% RSLogix 500 project COMPARATOR_BAK026.RSS, saved by version 8.30.00.16 %
PROJECT "UNTITLED"    % processor: Bul.1763 MicroLogix 1100 Series B %

PROGRAM FILES
  LAD 2   9 rungs

DATA FILES
  O0 OUTPUT  4 elements
  I1 INPUT  6 elements
  S2 STATUS  66 elements
  B3 BINARY  1 elements
  T4 TIMER  1 elements
  C5 COUNTER  1 elements
  R6 CONTROL  1 elements
  N7 INTEGER  1 elements
  F8 FLOAT  1 elements

LADDER 2
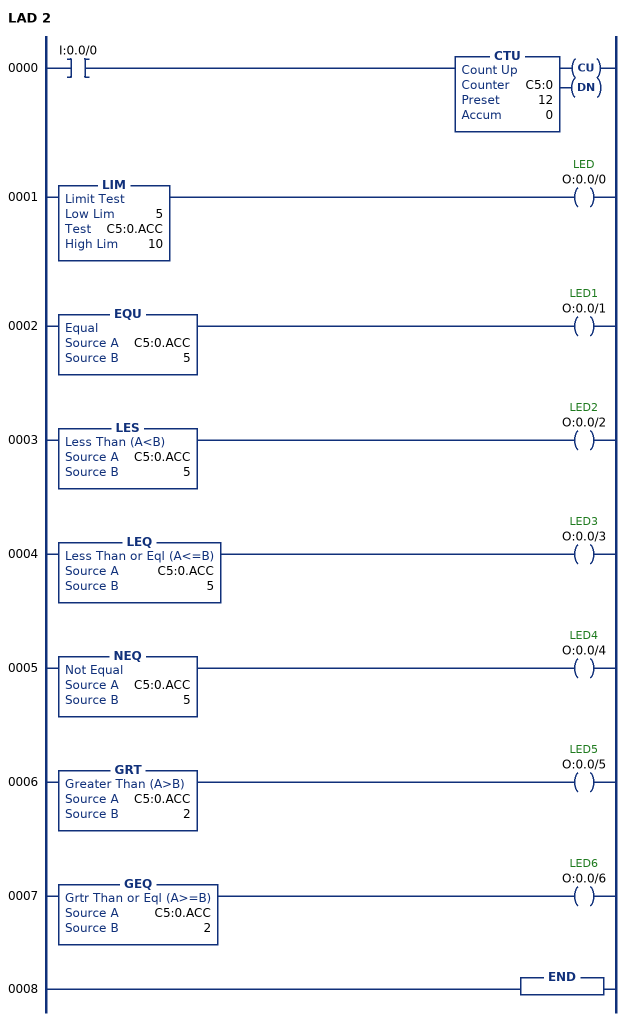
% Rung: 0 %
SOR XIC I:0.0/0 CTU C5:0 12 0 EOR
% Rung: 1 %
SOR LIM 5 C5:0.ACC 10 OTE O:0.0/0 EOR
%   O:0.0/0  "LED" %
% Rung: 2 %
SOR EQU C5:0.ACC 5 OTE O:0.0/1 EOR
%   O:0.0/1  "LED1" %
% Rung: 3 %
SOR LES C5:0.ACC 5 OTE O:0.0/2 EOR
%   O:0.0/2  "LED2" %
% Rung: 4 %
SOR LEQ C5:0.ACC 5 OTE O:0.0/3 EOR
%   O:0.0/3  "LED3" %
% Rung: 5 %
SOR NEQ C5:0.ACC 5 OTE O:0.0/4 EOR
%   O:0.0/4  "LED4" %
% Rung: 6 %  % edit flag set %
SOR GRT C5:0.ACC 2 OTE O:0.0/5 EOR
%   O:0.0/5  "LED5" %
% Rung: 7 %  % edit flag set %
SOR GEQ C5:0.ACC 2 OTE O:0.0/6 EOR
%   O:0.0/6  "LED6" %
% Rung: 8 %
SOR END EOR

DATA TABLE (non-zero values as saved)
DATA C5
% .PRE .ACC %
% C5:0 % 12 0
